Staubli VAL3: Form_Panel4P.pgx

public program Form_Panel4P(string x_sTitle, string x_sPanelTitle, num x_nItemCount, num& x_nSelectIndex, string x_sBottom)
  local num l_nNum
begin

//×××××××××××××××××××××××××××××××××××××××××××××××××
//×××××××××××××××××××××××××××××××××××××××××××××××××


x_nItemCount=max(0,x_nItemCount)

if x_nItemCount==0

  call Form_Panel(x_sTitle,x_sPanelTitle,x_nSelectIndex,x_sBottom)
  return
endIf


resize(sBuff,1,x_nItemCount)
for l_nNum=0 to x_nItemCount-1
//  if x_bList[l_nNum]
//    sBuff[l_nNum]=toString("",l_nNum+1)+"."+x_sList[l_nNum]
//  else
    sBuff[l_nNum]=toString("",l_nNum+1)+"."+"Point"
//  endIf
endFor
//*********************************************************
call Form_PanelList(x_sTitle,x_sPanelTitle,sBuff,x_nSelectIndex,x_sBottom)



end
